FUNCTION_BLOCK Kulbana
  (* Version 1.0, 2005-06-12, Goran Cengic, Chalmers *)
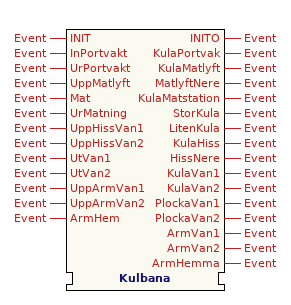
  EVENT_INPUT
    INIT;
    InPortvakt;
    UrPortvakt;
    UppMatlyft;
    Mat;
    UrMatning;
    UppHissVan1;
    UppHissVan2;
    UtVan1;
    UtVan2;
    UppArmVan1;
    UppArmVan2;
    ArmHem;
  END_EVENT
  EVENT_OUTPUT
    INITO;
    KulaPortvak;
    KulaMatlyft;
    MatlyftNere;
    KulaMatstation;
    StorKula;
    LitenKula;
    KulaHiss;
    HissNere;
    KulaVan1;
    KulaVan2;
    PlockaVan1;
    PlockaVan2;
    ArmVan1;
    ArmVan2;
    ArmHemma;
  END_EVENT
  VAR
    liten_kula : INT := 0;
  END_VAR
  EC_STATES
    START;
    INIT : -> INITO;
    STATE1 : PrintKulaPortvakt -> KulaPortvakt;
    STATE2 : PrintKulaMatlyft -> KulaMatlyft;
    STATE3 : PrintKulaMatstation -> KulaMatstation;
    STATE4 : PrintStorKula -> StorKula;
    STATE5 : PrintLitenKula -> LitenKula;
    STATE6 : PrintKulaHiss -> KulaHiss, -> MatlyftNere;
    STATE7 : PrintKulaVan1 -> KulaVan1;
    STATE8 : PrintKulaVan2 -> KulaVan2;
    STATE9 : PrintPlockaVan1 -> PlockaVan1, -> HissNere;
    STATE10 : PrintPlockaVan2 -> PlockaVan2, -> HissNere;
    STATE11 : PrintArmVan1 -> ArmVan1;
    STATE12 : PrintArmVan2 -> ArmVan2;
    STATE13 : PrintArmHemma -> ArmHemma;
  END_STATES
  EC_TRANSITIONS
    START TO INIT := INIT;
    INIT TO START := 1;
    START TO STATE1 := InPortvakt;
    STATE1 TO START := 1;
    START TO STATE2 := UrPortvakt;
    STATE2 TO START := 1;
    START TO STATE3 := UppMatlyft;
    STATE3 TO START := 1;
    START TO STATE4 := Mat AND (liten_kula MOD 3 = 0);
    STATE4 TO START := 1;
    START TO STATE5 := Mat AND (liten_kula MOD 3 > 0);
    STATE5 TO START := 1;
    START TO STATE6 := UrMatning;
    STATE6 TO START := 1;
    START TO STATE7 := UppHissVan1;
    STATE7 TO START := 1;
    START TO STATE8 := UppHissVan2;
    STATE8 TO START := 1;
    START TO STATE9 := UtVan1;
    STATE9 TO START := 1;
    START TO STATE10 := UtVan2;
    STATE10 TO START := 1;
    START TO STATE11 := UppArmVan1;
    STATE11 TO START := 1;
    START TO STATE12 := UppArmVan2;
    STATE12 TO START := 1;
    START TO STATE13 := ArmHem;
    STATE13 TO START := 1;
  END_TRANSITIONS
  ALGORITHM PrintKulaPortvakt IN Java:
System.out.println("KulaPortvakt");
  END_ALGORITHM
  ALGORITHM PrintKulaMatlyft IN Java:
System.out.println("KulaMatlyft");
  END_ALGORITHM
  ALGORITHM PrintKulaMatstation IN Java:
System.out.println("KulaMatstation");
  END_ALGORITHM
  ALGORITHM PrintStorKula IN Java:
liten_kula = liten_kula + 1;
		System.out.println("StorKula");
  END_ALGORITHM
  ALGORITHM PrintLitenKula IN Java:
liten_kula = liten_kula + 1;
		System.out.println("LitenKula");
  END_ALGORITHM
  ALGORITHM PrintKulaHiss IN Java:
System.out.println("KulaHiss");
  END_ALGORITHM
  ALGORITHM PrintKulaVan1 IN Java:
System.out.println("KulaVan1");
  END_ALGORITHM
  ALGORITHM PrintKulaVan2 IN Java:
System.out.println("KulaVan2");
  END_ALGORITHM
  ALGORITHM PrintPlockaVan1 IN Java:
System.out.println("PlockaVan1");
  END_ALGORITHM
  ALGORITHM PrintPlockaVan2 IN Java:
System.out.println("PlockaVan2");
  END_ALGORITHM
  ALGORITHM PrintArmVan1 IN Java:
System.out.println("ArmVan1");
  END_ALGORITHM
  ALGORITHM PrintArmVan2 IN Java:
System.out.println("ArmVan2");
  END_ALGORITHM
  ALGORITHM PrintArmHemma IN Java:
System.out.println("ArmHemma");
  END_ALGORITHM
END_FUNCTION_BLOCK
